// SIMATIC STEP 7 (V5.x) project PROJECT-PROFIBUS_en
// CPU: CPU 314(1)
// CPU: CPU 314(1)
// CPU: CPU 314(1)
// CPU: CPU 314(1)
// CPU: CPU 314(1)
// CPU: CPU 414-2 DP(1)
// CPU: CPU 414-2 DP(1)
// station: P_ADR_BUS
// station: Hardware
// station: FMS-Server S7 400-Stat.
// station: P_ADR_BUS
// station: Hardware
// station: SIMATIC 300-Station(1)
// station: P_ADR_BUS
// station: Hardware
// station: SIMATIC 300-Station(3)
// station: P_ADR_BUS
// station: Hardware
// station: SIMATIC 300 DP-Slave
// station: P_ADR_BUS
// station: Hardware
// station: FMS-Client S7 400-Stat.
// station: P_ADR_BUS
// station: Hardware
// station: SIMATIC 300-Station(2)
// station: P_ADR_BUS
// station: Hardware
// station: SIMATIC 300 DP-Master
// station: ISA_LOCAL_ADR_BUS
// program: S7 Programm (6)
// program: S7 Program (3)
// program: S7 Program(2)
// program: S7 Program (5)
// program: S7 Program (7)
// program: S7 Program (4)
// program: S7 Program(1)

SYMBOL_TABLE
"Index100 READ parameters"	DB 100	DB 100	// READ parameters
"Index101 READ parameters"	DB 101	DB 101	// READ parameters
"Index102 READ parameters"	DB 102	DB 102	// READ parameters
"Index100 WRITE parameter"	DB 200	DB 200	// WRITE parameters
"Index101 WRITE parameter"	DB 201	DB 201	// WRITE parameters
"Index102 WRITE parameter"	DB 202	DB 202	// WRITE parameters
"Index100 Variable dest"	DB 500	DB 500	// Variable destination
"Index101 Variable dest"	DB 501	DB 501	// Variable destination
"Index102 Variable dest"	DB 502	DB 502	// Variable destination
"Index100 Variable source"	DB 600	DB 600	// Variable source
"Index101 Variable source"	DB 601	DB 601	// Variable source
"Index102 Variable source"	DB 602	DB 602	// Variable source
"IDENT"	FB 2	FB 2	// FMS IDENT
"READ"	FB 3	FB 3	// Read function block for FMS services with SIMATIC NET CPs
"WRITE"	FB 6	FB 6	// Write function block for FMS services with SIMATIC NET CPs
"Index100 READ call"	FC 100	FC 100	// READ call
"Index101 READ call"	FC 101	FC 101	// READ call
"Index102 READ call"	FC 102	FC 102	// READ call
"Index100 WRITE call"	FC 200	FC 200	// WRITE call
"Index101 WRITE call"	FC 201	FC 201	// WRITE call
"Index102 WRITE call"	FC 202	FC 202	// WRITE call
"Compare Index 100"	FC 300	FC 300	// Compare index 100
"Error check"	M 0.0	BOOL	// Error check
"BSEND"	SFB 12	SFB 12	// Block-oriented send
"BRCV"	SFB 13	SFB 13	// Block-oriented receive
"BLKMOV"	SFC 20	SFC 20	// Direct word move
"TEST_DB"	SFC 24	SFC 24	// Debug data block
"CONTROL"	SFC 62	SFC 62	// Control status of a CFB instance
"observe Read/Write"	VAT 1		// Monitor read/write
"observe variables"	VAT 2		// Monitor variables
END_SYMBOL_TABLE

// FB 3: know-how protected block, not included

// FB 6: know-how protected block, not included

FUNCTION "Index100 READ call" : VOID	// FC 100
TITLE = CALL_READ
//This function illustrates an FMS communication job with the READ (FB3) function 
//block. A variable of the type integer is accessed.
VERSION : 0.1
BEGIN
NETWORK
TITLE = Read variable with index 100. 
//Read data access:   
//A variable with index 100 is read and entered in the destination data area 
//(here 
//DB500).
//Call parameters in DB 100.
//
//Job handling /job coordination:
//This job is only started when all other jobs have been completed. This means 
//that access to the variable is synchronized.
//The job is triggered by a signal edge at the REQ input. REQ is reset when the 
//job is completed or an error occurred. Following this, the signal is set again.
//If an error occurred, the error number can be read from the status word.
//*
//Only execute job when no other job is active.
      O     "Index100 WRITE parameter".Write_REQ;	//  REQ=1, WRITE is still active
      O     "Index101 READ parameters".Read_REQ;	//    REQ=1, READ is still active
      O     "Index101 WRITE parameter".Write_REQ;	//  REQ=1, WRITE is still active
      O     "Index102 READ parameters".Read_REQ;	//    REQ=1, READ is still active
      O     "Index102 WRITE parameter".Write_REQ;	//  REQ=1, WRITE is still active
      JC    ende;
//*
//Calling the READ job:                                       
//*
//*
//Query job status
//*
//*
//*
//Error handling
//*
      CALL  "READ" , DB 300 (
           DIX 0.0                  := "Index100 READ parameters".Read_REQ,
           DID 2                    := "Index100 READ parameters".Read_ID,
           DIW 6                    := W#16#1002,
           DIW 8                    := 7,
           DIW 10                   := 100,
           DID 12                   := P#DBX 6.0,
           DIW 16                   := W#16#1005,
           DIW 18                   := 1,
           DIW 20                   := 500,
           DID 22                   := P#DBX 0.0,
           DIX 26.0                 := "Index100 READ parameters".Read_NDR,
           DIX 26.1                 := "Index100 READ parameters".Read_Error,
           DIW 28                   := "Index100 READ parameters".Read_Status);	//  REQ=1 => Job active, query errors  /   REQ=1 => Job completed  /   Set REQ again /  Error=0 => No error occurred
      A     "Index100 READ parameters".Read_REQ;
//*
      JC    fehl;	// Error=1 => Error occurred 
      AN    "Index100 READ parameters".Read_REQ;	//Load error status
      S     "Index100 READ parameters".Read_REQ;	// Save in buffer
      JU    ende;	//   Reset REQ
fehl: AN    "Index100 READ parameters".Read_Error;
//*
//Query job status
//*
      JC    ok;	//  Done=0 => Job still active
      A     "Index100 READ parameters".Read_Error;
//*
      L     "Index100 READ parameters".Read_Status;	//  Done=1 => Job complete without error
      T     "Index100 READ parameters".Read_Statusmemory;	//  Reset REQ
//*
      R     "Index100 READ parameters".Read_REQ;
      JU    ende;
ok:   AN    "Index100 READ parameters".Read_NDR;
      JC    ende;
      A     "Index100 READ parameters".Read_NDR;
      R     "Index100 READ parameters".Read_REQ;
ende: BE;
END_FUNCTION

FUNCTION "Index101 READ call" : VOID	// FC 101
TITLE = CALL_READ
//The function illustrates an FMS communication job with the READ (FB3) function 
//block. A variable of the type array is accessed.
VERSION : 0.1
BEGIN
NETWORK
TITLE = Read variable with index 101. 
//Read data access:
//The variable with index 101 is read and entered in the destination data area 
//(here DB501). Call parameters in DB101.
//
//Job handling /job coordination:
//This job is only started when all other jobs have been completed. This means 
//that access to the variable is synchronized.
//The job is triggered by a signal edge at the REQ input. REQ is reset when the 
//job is completed or an error occurred. Following this, the signal is set again.
//If an error occurred, the error number can be read from the status word.
//
//*
// Only execute job when no other job is active.
//*
      O     "Index100 WRITE parameter".Write_REQ;	//  REQ=1, WRITE is still active
      O     "Index100 READ parameters".Read_REQ;	//    REQ=1, READ is still active
      O     "Index101 WRITE parameter".Write_REQ;	//  REQ=1, WRITE is still active
      O     "Index102 READ parameters".Read_REQ;	//    REQ=1, READ is still active
      O     "Index102 WRITE parameter".Write_REQ;	//  REQ=1, WRITE is still active
      JC    ende;
//*
//Calling the READ job:                                       
//*
//*
//Query job status
//*
//*
//*
//Error handling
//*
      CALL  "READ" , DB 301 (
           DIX 0.0                  := "Index101 READ parameters".Read_REQ,
           DID 2                    := "Index101 READ parameters".Read_ID,
           DIW 6                    := W#16#1002,
           DIW 8                    := 7,
           DIW 10                   := 101,
           DID 12                   := P#DBX 6.0,
           DIW 16                   := W#16#1002,
           DIW 18                   := 10,
           DIW 20                   := 501,
           DID 22                   := P#DBX 0.0,
           DIX 26.0                 := "Index101 READ parameters".Read_NDR,
           DIX 26.1                 := "Index101 READ parameters".Read_Error,
           DIW 28                   := "Index101 READ parameters".Read_Status);	//   REQ=1 => Job active, query errors /    REQ=1 => Job completed /    REQ neu setzten / Set REQ again /  Error=0 => No error occurred
      A     "Index101 READ parameters".Read_REQ;
//*
      JC    fehl;	// Error=1 => Error occurred
      AN    "Index101 READ parameters".Read_REQ;	// load error status
      S     "Index101 READ parameters".Read_REQ;	// Save in buffer
      JU    ende;	//   Reset REQ
fehl: AN    "Index101 READ parameters".Read_Error;
//*
//Query job status
//*
      JC    ok;	//  Done=0 => Job still active
      A     "Index101 READ parameters".Read_Error;
//*
      L     "Index101 READ parameters".Read_Status;	//  Done=1 => Job complete without error
      T     "Index101 READ parameters".Read_Statusspeicher;	//  Reset REQ
//*
      R     "Index101 READ parameters".Read_REQ;
      JU    ende;
ok:   AN    "Index101 READ parameters".Read_NDR;
      JC    ende;
      A     "Index101 READ parameters".Read_NDR;
      R     "Index101 READ parameters".Read_REQ;
ende: BE;
END_FUNCTION

FUNCTION "Index102 READ call" : VOID	// FC 102
TITLE = CALL_READ
//This function illustrates an FMS communication job with the READ (FB3) function 
//block. A variable of the type STRUCT is accessed.
VERSION : 0.1
BEGIN
NETWORK
TITLE = Read variable with index 102.
//Read data access:   
//A variable with index 102 is read and entered in the destination data area 
//(here 
//DB502). Call parameters in DB 100.
//
//Job handling /job coordination:
//This job is only started when all other jobs have been completed. This means 
//that access to the variable is synchronized.
//The job is triggered by a signal edge at the REQ input. REQ is reset when the 
//job is completed or an error occurred. Following this, the signal is set again.
//If an error occurred, the error number can be read from the status word.
//*
// Query whether other jobs still active
//*
      O     "Index100 READ parameters".Read_REQ;	//    REQ=1, READ is still active
      O     "Index100 WRITE parameter".Write_REQ;	//  REQ=1, WRITE is still active
      O     "Index101 READ parameters".Read_REQ;	//    REQ=1, READ is still active
      O     "Index101 WRITE parameter".Write_REQ;	//  REQ=1, WRITE is still active
      O     "Index102 WRITE parameter".Write_REQ;	//  REQ=1, WRITEis still active
      JC    ende;
//*
// Calling the READ job                                      
//*
//*
// Query the job status
//*
//*
//*
// Error handling
//*
      CALL  "READ" , DB 302 (
           DIX 0.0                  := "Index102 READ parameters".Read_REQ,
           DID 2                    := "Index102 READ parameters".Read_ID,
           DIW 6                    := W#16#1002,
           DIW 8                    := 7,
           DIW 10                   := 102,
           DID 12                   := P#DBX 6.0,
           DIW 16                   := W#16#1002,
           DIW 18                   := 18,
           DIW 20                   := 502,
           DID 22                   := P#DBX 0.0,
           DIX 26.0                 := "Index102 READ parameters".Read_NDR,
           DIX 26.1                 := "Index102 READ parameters".Read_Error,
           DIW 28                   := "Index102 READ parameters".Read_Status);	//   REQ=1 => Job active, query errors /    REQ=1 => Job completed /    Set REQ again /  Error=0 => No error occurred
      A     "Index102 READ parameters".Read_REQ;
//*
      JC    fehl;	//  Error=1 => Error occurred
      AN    "Index102 READ parameters".Read_REQ;	// Load error status
      S     "Index102 READ parameters".Read_REQ;	// Save in buffer
      JU    ende;	//  Reset REQ
fehl: AN    "Index102 READ parameters".Read_Error;
//*
// Query job status
//*
      JC    ok;	//  Done=0 => Job still active
      A     "Index102 READ parameters".Read_Error;
//*
      L     "Index102 READ parameters".Read_Status;	// Done=1 => Job complete without error
      T     "Index102 READ parameters".Read_Statusspeicher;	//   Reset REQ
//*
      R     "Index102 READ parameters".Read_REQ;
      JU    ende;
ok:   AN    "Index102 READ parameters".Read_NDR;
      JC    ende;
      A     "Index102 READ parameters".Read_NDR;
      R     "Index102 READ parameters".Read_REQ;
ende: BE;
END_FUNCTION

FUNCTION "Index100 WRITE call" : VOID	// FC 200
TITLE = CALL_WRITE
//This function illustrates an FMS communication job with the WRITE (FB6) 
//function 
//block. A variable of the type integer is accessed.
VERSION : 0.1
BEGIN
NETWORK
TITLE = Write var. with index 100 
//Write data access:   
//A variable with index 100 is written. It is taken from the source data area 
//(here DB600). Call parameters in DB200.
//
//Job handling /job coordination:
//This job is only started when all other jobs have been completed. This means 
//that access to the variable is synchronized.
//The job is triggered by a signal edge at the REQ input. REQ is reset when the 
//job is completed or an error occurred. Following this, the signal is set again.
//If an error occurred, the error number can be read from the status word.
//
//*  
// Query whether other jobs active
//*
      O     "Index100 READ parameters".Read_REQ;	//    REQ=1, WRITE is still active
      O     "Index101 READ parameters".Read_REQ;	//    REQ=1, READ is still active
      O     "Index101 WRITE parameter".Write_REQ;	//  REQ=1, WRITE is still active
      O     "Index102 READ parameters".Read_REQ;	//    REQ=1, READ is still active
      O     "Index102 WRITE parameter".Write_REQ;	//  REQ=1, WRITE is still active
      JC    ende;
//*
// Calling the write job               
//*
//*
// Query the job status
//*
//*
// *
// Error handling
//*
      CALL  "WRITE" , DB 400 (
           DIX 0.0                  := "Index100 WRITE parameter".Write_REQ,
           DID 2                    := "Index100 WRITE parameter".Write_ID,
           DIW 6                    := W#16#1002,
           DIW 8                    := 7,
           DIW 10                   := 200,
           DID 12                   := P#DBX 6.0,
           DIW 16                   := W#16#1005,
           DIW 18                   := 1,
           DIW 20                   := 600,
           DID 22                   := P#DBX 0.0,
           DIX 26.0                 := "Index100 WRITE parameter".Write_Done,
           DIX 26.1                 := "Index100 WRITE parameter".Write_Error,
           DIW 28                   := "Index100 WRITE parameter".Write_Status);	//    REQ=1 => Job active, query errors /     REQ=1 => Job completed  /     Set REQ again /   Error=0 => No error occurred
      A     "Index100 WRITE parameter".Write_REQ;
//*
      JC    fehl;	//  Error=1 => Error occurred
      AN    "Index100 WRITE parameter".Write_REQ;	// Load error status
      S     "Index100 WRITE parameter".Write_REQ;	// Save in buffer
      JU    ende;	//    Reset REQ
fehl: AN    "Index100 WRITE parameter".Write_Error;
//*
// Query job status 
//*
      JC    ok;	//   Done=0 => Job still active
      A     "Index100 WRITE parameter".Write_Error;
//*
      L     "Index100 WRITE parameter".Write_Status;	//   Done=1 => Job complete without error
      T     "Index100 WRITE parameter".Write_Statusspeicher;	//     / Reset REQ
//*
      R     "Index100 WRITE parameter".Write_REQ;
      JU    ende;
ok:   AN    "Index100 WRITE parameter".Write_Done;
      JC    ende;
      A     "Index100 WRITE parameter".Write_Done;
      R     "Index100 WRITE parameter".Write_REQ;
ende: BE;
END_FUNCTION

FUNCTION "Index101 WRITE call" : VOID	// FC 201
TITLE = CALL_WRITE
//This function illustrates an FMS communication job with the WRITE (FB6) 
//function 
//block. A variable of the type ARRAY is accessed.
//
VERSION : 0.1
BEGIN
NETWORK
TITLE = Write var with index 101. 
//Write data access:   
//A variable with index 100 is written. It is taken from the source data area 
//(here DB601). Call parameters in DB201.
//
//Job handling /job coordination:
//This job is only started when all other jobs have been completed. This means 
//that access to the variable is synchronized.
//The job is triggered by a signal edge at the REQ input. REQ is reset when the 
//job is completed or an error occurred. Following this, the signal is set 
//again.
//If an error occurred, the error number can be read from the status word.
//*  
// Query whether other jobs still active
//*
      O     "Index100 READ parameters".Read_REQ;	//    REQ=1, WRITE is still active
      O     "Index100 WRITE parameter".Write_REQ;	//  REQ=1, WRITE is still active
      O     "Index101 READ parameters".Read_REQ;	//    REQ=1, READ is still active
      O     "Index102 READ parameters".Read_REQ;	//    REQ=1, READ is still active
      O     "Index102 WRITE parameter".Write_REQ;	//  REQ=1, WRITE is still active
      JC    ende;
//*
// Calling the write job               
//*
//*
// Query job status
//*
//*
// *
// Error handling
//*
      CALL  "WRITE" , DB 401 (
           DIX 0.0                  := "Index101 WRITE parameter".Write_REQ,
           DID 2                    := "Index101 WRITE parameter".Write_ID,
           DIW 6                    := W#16#1002,
           DIW 8                    := 7,
           DIW 10                   := 201,
           DID 12                   := P#DBX 6.0,
           DIW 16                   := W#16#1002,
           DIW 18                   := 10,
           DIW 20                   := 601,
           DID 22                   := P#DBX 0.0,
           DIX 26.0                 := "Index101 WRITE parameter".Write_Done,
           DIX 26.1                 := "Index101 WRITE parameter".Write_Error,
           DIW 28                   := "Index101 WRITE parameter".Write_Status);	//    REQ=1 => Job active, query errors  /     REQ=1 => Job completed   /     Set REQ again /    Error=0 => No error occurred
      A     "Index101 WRITE parameter".Write_REQ;
//*
      JC    fehl;	//  Error=1 => Error occurred
      AN    "Index101 WRITE parameter".Write_REQ;	// Load error status
      S     "Index101 WRITE parameter".Write_REQ;	// Save in buffer
      JU    ende;	//    Reset REQ
fehl: AN    "Index101 WRITE parameter".Write_Error;
//*
// Query job status
//*
      JC    ok;	//   Done=0 => Job still active
      A     "Index101 WRITE parameter".Write_Error;
//*
      L     "Index101 WRITE parameter".Write_Status;	//   Done=1 => Job complete without error
      T     "Index101 WRITE parameter".Write_Statusspeicher;	//    Reset REQ
//*
      R     "Index101 WRITE parameter".Write_REQ;
      JU    ende;
ok:   AN    "Index101 WRITE parameter".Write_Done;
      JC    ende;
      A     "Index101 WRITE parameter".Write_Done;
      R     "Index101 WRITE parameter".Write_REQ;
ende: BE;
END_FUNCTION

FUNCTION "Index102 WRITE call" : VOID	// FC 202
TITLE = CALL_WRITE
//This function illustrates an FMS communication job with the WRITE (FB6) 
//function 
//block. A variable of the type STRUCT is accessed.
//
VERSION : 0.1
BEGIN
NETWORK
TITLE = Write var with index 102.
//Write data access:   
//A variable with index 102 is written. It is taken from the source data area 
//(here DB602). Call parameters in DB202.
//
//Job handling /job coordination:
//This job is only started when all other jobs have been completed. This means 
//that access to the variable is synchronized.
//The job is triggered by a signal edge at the REQ input. REQ is reset when the 
//job is completed or an error occurred. Following this, the signal is set again.
//If an error occurred, the error number can be read from the status word.
//
//
//*  
// Query whether other jobs active
//*       
      O     "Index100 READ parameters".Read_REQ;	//    REQ=1, READ is still active
      O     "Index100 WRITE parameter".Write_REQ;	//  REQ=1, WRITE is still active
      O     "Index101 READ parameters".Read_REQ;	//    REQ=1, REA is still active
      O     "Index101 WRITE parameter".Write_REQ;	//  REQ=1, WRITE is still active
      O     "Index102 READ parameters".Read_REQ;	//    REQ=1, REA is still active
      JC    ende;
//*
// Calling the write job               
//*
//*
// Query job status
//*
//*
// *
// Error handling
//*
      CALL  "WRITE" , DB 402 (
           DIX 0.0                  := "Index102 WRITE parameter".Write_REQ,
           DID 2                    := "Index102 WRITE parameter".Write_ID,
           DIW 6                    := W#16#1002,
           DIW 8                    := 7,
           DIW 10                   := 202,
           DID 12                   := P#DBX 6.0,
           DIW 16                   := W#16#1002,
           DIW 18                   := 18,
           DIW 20                   := 602,
           DID 22                   := P#DBX 0.0,
           DIX 26.0                 := "Index102 WRITE parameter".Write_Done,
           DIX 26.1                 := "Index102 WRITE parameter".Write_Error,
           DIW 28                   := "Index102 WRITE parameter".Write_Status);	//    REQ=1 => Job active, query errors /     REQ=1 => Job completed /     Set REQ again /   Error=0 => No error occurred
      A     "Index102 WRITE parameter".Write_REQ;
//*
      JC    fehl;	//  Error=1 => Error occurred
      AN    "Index102 WRITE parameter".Write_REQ;	// Load error status
      S     "Index102 WRITE parameter".Write_REQ;	// Save in buffer
      JU    ende;	//    Reset REQ
fehl: AN    "Index102 WRITE parameter".Write_Error;
//*
// Query job status 
//*
      JC    ok;	//   Done=0 => Job still active
      A     "Index102 WRITE parameter".Write_Error;
//*
      L     "Index102 WRITE parameter".Write_Status;	//   Done=1 => Job complete without error
      T     "Index102 WRITE parameter".Write_Statusspeicher;	//    Reset REQ
//*
      R     "Index102 WRITE parameter".Write_REQ;
      JU    ende;
ok:   AN    "Index102 WRITE parameter".Write_Done;
      JC    ende;
      A     "Index102 WRITE parameter".Write_Done;
      R     "Index102 WRITE parameter".Write_REQ;
ende: BE;
END_FUNCTION

FUNCTION "Compare Index 100" : VOID	// FC 300
//This function simulates a signal or value change and checks the write or read 
//function via the FMS connection. 
VERSION : 0.1
BEGIN
NETWORK
TITLE = Error check
//After writing and reading index 100, the values are compared to check that they 
//match. Afterwards the variable is incremented by one.
//
//*
      L     "Index100 Variable dest".Index_100;
      L     "Index100 Variable source".Index_100;
      ==I;
      JC    inkr;
//*
// Set memory bit 0.0 if the source and destination do not match.
//*
      S     "Error check";
//*
// Increment variable with index 100 by one
//*
inkr: L     "Index100 Variable source".Index_100;
      +     1;
      T     "Index100 Variable source".Index_100;
      R     "Error check";
//*
      BE;
END_FUNCTION

DATA_BLOCK "Index100 READ parameters"	// DB 100
VERSION : 0.1
  STRUCT
   Read_REQ : BOOL ;
   Read_ID : DWORD  := DW#16#10001;
   Read_VAR_Index : STRING  [5 ] := '<100>';
   Read_NDR : BOOL ;
   Read_Error : BOOL ;
   Read_Status : WORD ;
   Read_Statusmemory : WORD ;
  END_STRUCT ;	
BEGIN
   Read_ID := DW#16#10001;
   Read_VAR_Index := '<100>';
END_DATA_BLOCK

DATA_BLOCK "Index101 READ parameters"	// DB 101
VERSION : 0.1
  STRUCT
   Read_REQ : BOOL ;
   Read_ID : DWORD  := DW#16#10001;
   Read_VAR_Index : STRING  [5 ] := '<101>';
   Read_NDR : BOOL ;
   Read_Error : BOOL ;
   Read_Status : WORD ;
   Read_Statusspeicher : WORD ;
  END_STRUCT ;	
BEGIN
   Read_ID := DW#16#10001;
   Read_VAR_Index := '<101>';
END_DATA_BLOCK

DATA_BLOCK "Index102 READ parameters"	// DB 102
VERSION : 0.1
  STRUCT
   Read_REQ : BOOL ;
   Read_ID : DWORD  := DW#16#10001;
   Read_VAR_Index : STRING  [5 ] := '<102>';
   Read_NDR : BOOL ;
   Read_Error : BOOL ;
   Read_Status : WORD ;
   Read_Statusspeicher : WORD ;
  END_STRUCT ;	
BEGIN
   Read_ID := DW#16#10001;
   Read_VAR_Index := '<102>';
END_DATA_BLOCK

DATA_BLOCK "Index100 WRITE parameter"	// DB 200
VERSION : 0.1
  STRUCT
   Write_REQ : BOOL ;
   Write_ID : DWORD  := DW#16#10001;
   Write_VAR_Index : STRING  [5 ] := '<100>';
   Write_Done : BOOL ;
   Write_Error : BOOL ;
   Write_Status : WORD ;
   Write_Statusspeicher : WORD ;
   Write_VAR_Index1 : STRING  [5 ] := '<100>';
   tdmset : BYTE ;
  END_STRUCT ;	
BEGIN
   Write_ID := DW#16#10001;
   Write_VAR_Index := '<100>';
   Write_VAR_Index1 := '<100>';
END_DATA_BLOCK

DATA_BLOCK "Index101 WRITE parameter"	// DB 201
VERSION : 0.1
  STRUCT
   Write_REQ : BOOL ;
   Write_ID : DWORD  := DW#16#10001;
   Write_VAR_Index : STRING  [5 ] := '<101>';
   Write_Done : BOOL ;
   Write_Error : BOOL ;
   Write_Status : WORD ;
   Write_Statusspeicher : WORD ;
  END_STRUCT ;	
BEGIN
   Write_ID := DW#16#10001;
   Write_VAR_Index := '<101>';
END_DATA_BLOCK

DATA_BLOCK "Index102 WRITE parameter"	// DB 202
VERSION : 0.1
  STRUCT
   Write_REQ : BOOL ;
   Write_ID : DWORD  := DW#16#10001;
   Write_VAR_Index : STRING  [5 ] := '<102>';
   Write_Done : BOOL ;
   Write_Error : BOOL ;
   Write_Status : WORD ;
   Write_Statusspeicher : WORD ;
  END_STRUCT ;	
BEGIN
   Write_ID := DW#16#10001;
   Write_VAR_Index := '<102>';
END_DATA_BLOCK

DATA_BLOCK DB 300
AUTHOR : SIMATIC
FAMILY : CP_400
VERSION : 0.0
"READ"
BEGIN
END_DATA_BLOCK

DATA_BLOCK DB 301
AUTHOR : SIMATIC
FAMILY : CP_400
VERSION : 0.0
"READ"
BEGIN
END_DATA_BLOCK

DATA_BLOCK DB 302
AUTHOR : SIMATIC
FAMILY : CP_400
VERSION : 0.0
"READ"
BEGIN
END_DATA_BLOCK

DATA_BLOCK DB 400
AUTHOR : SIMATIC
FAMILY : CP_400
VERSION : 0.0
"WRITE"
BEGIN
END_DATA_BLOCK

DATA_BLOCK DB 401
AUTHOR : SIMATIC
FAMILY : CP_400
VERSION : 0.0
"WRITE"
BEGIN
END_DATA_BLOCK

DATA_BLOCK DB 402
AUTHOR : SIMATIC
FAMILY : CP_400
VERSION : 0.0
"WRITE"
BEGIN
END_DATA_BLOCK

DATA_BLOCK "Index100 Variable dest"	// DB 500
VERSION : 0.1
  STRUCT
   Index_100 : INT ;
  END_STRUCT ;	
BEGIN
END_DATA_BLOCK

DATA_BLOCK "Index101 Variable dest"	// DB 501
VERSION : 0.1
  STRUCT
   Index_101 : ARRAY  [1 .. 10 ] OF BYTE ;
  END_STRUCT ;	
BEGIN
END_DATA_BLOCK

DATA_BLOCK "Index102 Variable dest"	// DB 502
VERSION : 0.1
  STRUCT
   Index_102 : STRUCT
    Subindex_1 : BOOL ;
    Subindex_2 : STRING  [8 ];
    Subindex_3 : CHAR ;
    Subindex_4 : DINT ;
   END_STRUCT ;
  END_STRUCT ;	
BEGIN
   Index_102.Subindex_3 := ' ';
END_DATA_BLOCK

DATA_BLOCK "Index100 Variable source"	// DB 600
VERSION : 0.1
  STRUCT
   Index_100 : INT ;
  END_STRUCT ;	
BEGIN
END_DATA_BLOCK

DATA_BLOCK "Index101 Variable source"	// DB 601
VERSION : 0.1
  STRUCT
   Index_101 : ARRAY  [1 .. 10 ] OF BYTE ;
  END_STRUCT ;	
BEGIN
END_DATA_BLOCK

DATA_BLOCK "Index102 Variable source"	// DB 602
VERSION : 0.1
  STRUCT
   Index_102 : STRUCT
    Subindex_1 : BOOL ;
    Subindex_2 : STRING  [8 ] := 'Hello!!!';
    Subindex_3 : CHAR ;
    Subindex_4 : DINT ;
   END_STRUCT ;
  END_STRUCT ;	
BEGIN
   Index_102.Subindex_2 := 'Andreas!';
   Index_102.Subindex_3 := ' ';
END_DATA_BLOCK

ORGANIZATION_BLOCK OB 1
//Functions (FC100..FC300) in which FMS communication jobs are sent are called in 
//this block. The FCs are designed so that a coordinated sequence is guaranteed.
//(For the symbolic declaration, refer to the entries in the symbol table for 
//this 
//CPU.)
VERSION : 0.1
VAR_TEMP
  OB1_EV_CLASS : BYTE ;	//Bits 0-3 = 1 (Coming event), Bits 4-7 = 1 (Event class 1)
  OB1_SCAN_1 : BYTE ;	//1 (Cold restart scan 1 of OB 1), 3 (Scan 2-n of OB 1)
  OB1_PRIORITY : BYTE ;	//1 (Priority of 1 is lowest)
  OB1_OB_NUMBR : BYTE ;	//1 (Organization block 1, OB1)
  OB1_RESERVED_1 : BYTE ;	//Reserved for system
  OB1_RESERVED_2 : BYTE ;	//Reserved for system
  OB1_PREV_CYCLE : INT ;	//Cycle time of previous OB1 scan (milliseconds)
  OB1_MIN_CYCLE : INT ;	//Minimum cycle time of OB1 (milliseconds)
  OB1_MAX_CYCLE : INT ;	//Maximum cycle time of OB1 (milliseconds)
  OB1_DATE_TIME : DATE_AND_TIME ;	//Date and time OB1 started
END_VAR
BEGIN
NETWORK
TITLE =
//Write and read jobs are called sequentially.
      CALL  "Index100 READ call";
//*
      CALL  "Compare Index 100";
//*
      CALL  "Index100 WRITE call";
//*
      CALL  "Index101 READ call";
//*
      CALL  "Index101 WRITE call";
//*
      CALL  "Index102 READ call";
//*
      CALL  "Index102 WRITE call";
END_ORGANIZATION_BLOCK

ORGANIZATION_BLOCK OB 100
VERSION : 0.1
VAR_TEMP
  OB100_EV_CLASS : BYTE ;	//16#13, Event class 1, Entering event state, Event logged in diagnostic buffer
  OB100_STRTUP : BYTE ;	//16#81/82/83/84 Method of startup
  OB100_PRIORITY : BYTE ;	//27 (Priority of 1 is lowest)
  OB100_OB_NUMBR : BYTE ;	//100 (Organization block 100, OB100)
  OB100_RESERVED_1 : BYTE ;	//Reserved for system
  OB100_RESERVED_2 : BYTE ;	//Reserved for system
  OB100_STOP : WORD ;	//Event that caused CPU to stop (16#4xxx)
  OB100_STRT_INFO : DWORD ;	//Information on how system started
  OB100_DATE_TIME : DATE_AND_TIME ;	//Date and time OB100 started
END_VAR
BEGIN
NETWORK
TITLE =
      L     0;
      T     "Index100 Variable dest".Index_100;
      BE;
END_ORGANIZATION_BLOCK

SYMBOL_TABLE
"DP_SEND"	FC 1	FC 1	// DP SEND
"DP_RECV"	FC 2	FC 2	// DP RECEIVE
"DP_DIAG"	FC 3	FC 3	// DP DIAGNOSE
"DP_CTRL"	FC 4	FC 4	// DP CONTROL
"STP"	SFC 46	SFC 46	// Change the CPU to STOP
"WR_REC"	SFC 58	SFC 58	// Write Data Record
"RD_REC"	SFC 59	SFC 59	// Read a Data Record
END_SYMBOL_TABLE

// FC 1: know-how protected block, not included

// FC 2: know-how protected block, not included

// FC 3: know-how protected block, not included

// FC 4: know-how protected block, not included

FUNCTION FC 29 : VOID
TITLE = running light
VERSION : 0.1
BEGIN
NETWORK
TITLE =
      A     T 4;	//time downwards
      JC    runt;
st_1: A     M 40.1;	//start timer 3
      L     S5T#3S;	//LED upwards 3 sec.
      SE    T 3;
      A     T 3;
      R     M 40.1;
      JC    hoch;	//jump to upwards
      AN    T 3;
      S     M 40.1;
      S     M 40.2;
runt: A     M 40.2;	//start timer 4
      L     S5T#3S;	//LED downwards 3 sec.
      SE    T 4;
      A     T 4;
      R     M 40.2;
      AN    T 4;
      S     M 40.2;
      JC    st_1;
      A     M 40.0;
      L     S5T#100MS;
      SE    T 1;
      A     T 1;
      R     M 40.0;
      A     T 1;
      JC    weit;
      AN    T 1;
      S     M 40.0;
      L     MW 70;
      L     0;
      <>D;
      JC    los1;
      TAK;
      +     1;
      T     MW 70;
      T     DB30.DBW 1;
      BEU;
los1: L     MW 70;
      L     2;
      *D;
      T     MW 70;
      T     DB30.DBW 1;
      L     L#32768;
      <>D;
      BEC;
      L     0;
      T     MW 70;
weit: BEU;
hoch: A     M 40.3;
      L     S5T#100MS;
      SE    T 1;
      A     T 1;
      R     M 40.3;
      A     T 1;
      JC    weit;
      AN    T 1;
      S     M 40.3;
      L     MW 70;
      L     0;
      <>D;
      JC    los2;
      TAK;
      +     L#32768;
      T     MW 70;
      T     DB30.DBW 1;
      BEU;
los2: L     MW 70;
      L     2;
      /D;
      T     MW 70;
      T     DB30.DBW 1;
      L     1;
      <>D;
      BEC;
      L     0;
      T     MW 70;
      BE;
END_FUNCTION

ORGANIZATION_BLOCK OB 1
TITLE = co-ordination DP-Slave
//Co-ordination of the program sequence.
VERSION : 0.1
VAR_TEMP
  OB1_EV_CLASS : BYTE ;	//Bits 0-3 = 1 (Coming event), Bits 4-7 = 1 (Event class 1)
  OB1_SCAN_1 : BYTE ;	//1 (Cold restart scan 1 of OB 1), 3 (Scan 2-n of OB 1)
  OB1_PRIORITY : BYTE ;	//1 (Priority of 1 is lowest)
  OB1_OB_NUMBR : BYTE ;	//1 (Organization block 1, OB1)
  OB1_RESERVED_1 : BYTE ;	//Reserved for system
  OB1_RESERVED_2 : BYTE ;	//Reserved for system
  OB1_PREV_CYCLE : INT ;	//Cycle time of previous OB1 scan (milliseconds)
  OB1_MIN_CYCLE : INT ;	//Minimum cycle time of OB1 (milliseconds)
  OB1_MAX_CYCLE : INT ;	//Maximum cycle time of OB1 (milliseconds)
  OB1_DATE_TIME : DATE_AND_TIME ;	//Date and time OB1 started
END_VAR
BEGIN
NETWORK
TITLE =
      CALL  "DP_RECV" (
           $1                       := 272,
           $2                       := P#DB10.DBX 0.0 BYTE 10,
           $3                       := P#M 1.0,
           $4                       := M 1.1,
           $5                       := P#M 200.0,
           $6                       := P#M 202.0);	//Call DP_RECV
      L     DB10.DBW 0;	//output for simulation module
      T     QW 0;
      T     DB11.DBW 0;	//data for confirmation
      CALL  "DP_SEND" (
           $1                       := 272,
           $2                       := P#DB11.DBX 0.0 BYTE 10,
           $3                       := M 1.2,
           $4                       := M 1.3,
           $5                       := P#M 104.0);	//Call DP_SEND
      BE;
END_ORGANIZATION_BLOCK

ORGANIZATION_BLOCK OB 100
TITLE = create DB
//Creation of data blocks DB10 and DB11. The process values are saved in these 
//data blocks.
VERSION : 0.0
VAR_TEMP
  OB100_EV_CLASS : BYTE ;	//16#13, Event class 1, Entering event state, Event logged in diagnostic buffer
  OB100_STRTUP : BYTE ;	//16#81/82/83/84 Method of startup
  OB100_PRIORITY : BYTE ;	//27 (Priority of 1 is lowest)
  OB100_OB_NUMBR : BYTE ;	//100 (Organization block 100, OB100)
  OB100_RESERVED_1 : BYTE ;	//Reserved for system
  OB100_RESERVED_2 : BYTE ;	//Reserved for system
  OB100_STOP : WORD ;	//Event that caused CPU to stop (16#4xxx)
  OB100_STRT_INFO : DWORD ;	//Information on how system started
  OB100_DATE_TIME : DATE_AND_TIME ;	//Date and time OB100 started
END_VAR
BEGIN
NETWORK
TITLE =
      L     10;
      T     MW 20;
      L     11;
      T     MW 22;
      L     300;
      T     MW 24;
      CALL  SFC 22 (
           LOW_LIMIT                := MW 20,
           UP_LIMIT                 := MW 22,
           COUNT                    := MW 24,
           RET_VAL                  := MW 26,
           DB_NUMBER                := MW 26);
      CALL  SFC 22 (
           LOW_LIMIT                := MW 20,
           UP_LIMIT                 := MW 22,
           COUNT                    := MW 24,
           RET_VAL                  := MW 26,
           DB_NUMBER                := MW 28);
      BE;
END_ORGANIZATION_BLOCK

SYMBOL_TABLE
"AG_SEND"	FC 5	FC 5	// AG SEND
"AG_RECV"	FC 6	FC 6	// AG RECEIVE
END_SYMBOL_TABLE

// FC 5: know-how protected block, not included

// FC 6: know-how protected block, not included

FUNCTION FC 29 : VOID
TITLE = handling of the process data
//A data word is incremented and decremented cyclically. The time interval for 
//incrementing and decrementing is 3 seconds.
VERSION : 0.1
BEGIN
NETWORK
TITLE =
      A     T 4;	//time downwards
      JC    runt;
st_1: A     M 40.1;	//start timer 3
      L     S5T#3S;	//LED upwards 3 sec
      SE    T 3;
      A     T 3;
      R     M 40.1;
      JC    hoch;	//jump for upwards
      AN    T 3;
      S     M 40.1;
      S     M 40.2;
runt: A     M 40.2;	//start timer 4
      L     S5T#3S;	//LED downwards 3 sec
      SE    T 4;
      A     T 4;
      R     M 40.2;
      AN    T 4;
      S     M 40.2;
      JC    st_1;
      A     M 40.0;
      L     S5T#100MS;
      SE    T 1;
      A     T 1;
      R     M 40.0;
      A     T 1;
      JC    weit;
      AN    T 1;
      S     M 40.0;
      L     MW 70;
      L     0;
      <>D;
      JC    los1;
      TAK;
      +     1;
      T     MW 70;
      T     DB30.DBW 1;
      BEU;
los1: L     MW 70;
      L     2;
      *D;
      T     MW 70;
      T     DB30.DBW 1;
      L     L#32768;
      <>D;
      BEC;
      L     0;
      T     MW 70;
weit: BEU;
hoch: A     M 40.3;
      L     S5T#100MS;
      SE    T 1;
      A     T 1;
      R     M 40.3;
      A     T 1;
      JC    weit;
      AN    T 1;
      S     M 40.3;
      L     MW 70;
      L     0;
      <>D;
      JC    los2;
      TAK;
      +     L#32768;
      T     MW 70;
      T     DB30.DBW 1;
      BEU;
los2: L     MW 70;
      L     2;
      /D;
      T     MW 70;
      T     DB30.DBW 1;
      L     1;
      <>D;
      BEC;
      L     0;
      T     MW 70;
      BE;
END_FUNCTION

FUNCTION FC 30 : VOID
TITLE = Senden
//Sends data via FDL-connection with ID=1.
//Starting at byte 1 from DB30, 4 bytes are going to send.
VERSION : 0.0
BEGIN
NETWORK
TITLE =
      O     M 50.0;
      ON    M 50.0;
      S     M 50.0;
      CALL  "AG_SEND" (
           $1                       := P#M 50.0,
           $2                       := 1,
           $3                       := 272,
           $4                       := P#DB30.DBX 1.0 BYTE 240,
           $5                       := 4,
           $6                       := M 1.2,
           $7                       := M 1.3,
           $8                       := P#M 200.0);	//AG_SEND
      BE;
END_FUNCTION

FUNCTION FC 31 : VOID
TITLE = Receive
//Station 1
//
//Receives data via FDL-connection with ID=1.
//Data are accepted in DB31.
VERSION : 0.0
BEGIN
NETWORK
TITLE =
      CALL  "AG_RECV" (
           $1                       := 1,
           $2                       := 272,
           $3                       := P#DB31.DBX 1.0 BYTE 240,
           $4                       := P#M 1.0,
           $5                       := M 1.1,
           $6                       := P#M 202.0,
           $7                       := P#M 10.0);	//AG_RECV
      L     DB31.DBW 1;
      T     QW 0;
      BE;
END_FUNCTION

ORGANIZATION_BLOCK OB 1
TITLE = co-ordination
//Co-ordination of the program sequence.
VERSION : 0.1
VAR_TEMP
  OB1_EV_CLASS : BYTE ;	//Bits 0-3 = 1 (Coming event), Bits 4-7 = 1 (Event class 1)
  OB1_SCAN_1 : BYTE ;	//1 (Cold restart scan 1 of OB 1), 3 (Scan 2-n of OB 1)
  OB1_PRIORITY : BYTE ;	//1 (Priority of 1 is lowest)
  OB1_OB_NUMBR : BYTE ;	//1 (Organization block 1, OB1)
  OB1_RESERVED_1 : BYTE ;	//Reserved for system
  OB1_RESERVED_2 : BYTE ;	//Reserved for system
  OB1_PREV_CYCLE : INT ;	//Cycle time of previous OB1 scan (milliseconds)
  OB1_MIN_CYCLE : INT ;	//Minimum cycle time of OB1 (milliseconds)
  OB1_MAX_CYCLE : INT ;	//Maximum cycle time of OB1 (milliseconds)
  OB1_DATE_TIME : DATE_AND_TIME ;	//Date and time OB1 started
END_VAR
BEGIN
NETWORK
TITLE =
      CALL  FC 29;
      CALL  FC 30;
      CALL  FC 31;
      BE;
END_ORGANIZATION_BLOCK

ORGANIZATION_BLOCK OB 100
TITLE = Create DB
//Creation of data blocks DB30/DB31 with length 350 byte. The process values are 
//saved 
//in these data blocks.
VERSION : 0.0
VAR_TEMP
  OB100_EV_CLASS : BYTE ;	//16#13, Event class 1, Entering event state, Event logged in diagnostic buffer
  OB100_STRTUP : BYTE ;	//16#81/82/83/84 Method of startup
  OB100_PRIORITY : BYTE ;	//27 (Priority of 1 is lowest)
  OB100_OB_NUMBR : BYTE ;	//100 (Organization block 100, OB100)
  OB100_RESERVED_1 : BYTE ;	//Reserved for system
  OB100_RESERVED_2 : BYTE ;	//Reserved for system
  OB100_STOP : WORD ;	//Event that caused CPU to stop (16#4xxx)
  OB100_STRT_INFO : DWORD ;	//Information on how system started
  OB100_DATE_TIME : DATE_AND_TIME ;	//Date and time OB100 started
END_VAR
BEGIN
NETWORK
TITLE =
      L     30;
      T     MW 22;
      L     31;
      T     MW 24;
      L     350;
      T     MW 26;
      CALL  SFC 22 (
           LOW_LIMIT                := MW 22,
           UP_LIMIT                 := MW 24,
           COUNT                    := MW 26,
           RET_VAL                  := MW 28,
           DB_NUMBER                := MW 30);
      BE;
END_ORGANIZATION_BLOCK

SYMBOL_TABLE
"AG_SEND"	FC 5	FC 5	// AG SEND
"AG_RECV"	FC 6	FC 6	// AG RECEIVE
END_SYMBOL_TABLE

// FC 5: know-how protected block, not included

// FC 6: know-how protected block, not included

FUNCTION FC 29 : VOID
TITLE = handling of the process data
//A data word is incremented and decremented cyclically. The time interval for 
//incrementing and decrementing is 3 seconds.
VERSION : 0.1
BEGIN
NETWORK
TITLE =
      A     T 4;	//Time downwards
      JC    runt;
st_1: A     M 40.1;	//start timer 3
      L     S5T#3S;	//LED upwards 3 sec
      SE    T 3;
      A     T 3;
      R     M 40.1;
      JC    hoch;	//jump for upwards
      AN    T 3;
      S     M 40.1;
      S     M 40.2;
runt: A     M 40.2;	//start für timer 4
      L     S5T#3S;	//LED downwards 3 sec
      SE    T 4;
      A     T 4;
      R     M 40.2;
      AN    T 4;
      S     M 40.2;
      JC    st_1;
      A     M 40.0;
      L     S5T#100MS;
      SE    T 1;
      A     T 1;
      R     M 40.0;
      A     T 1;
      JC    weit;
      AN    T 1;
      S     M 40.0;
      L     MW 70;
      L     0;
      <>D;
      JC    los1;
      TAK;
      +     1;
      T     MW 70;
      T     DB30.DBW 1;
      BEU;
los1: L     MW 70;
      L     2;
      *D;
      T     MW 70;
      T     DB30.DBW 1;
      L     L#32768;
      <>D;
      BEC;
      L     0;
      T     MW 70;
weit: BEU;
hoch: A     M 40.3;
      L     S5T#100MS;
      SE    T 1;
      A     T 1;
      R     M 40.3;
      A     T 1;
      JC    weit;
      AN    T 1;
      S     M 40.3;
      L     MW 70;
      L     0;
      <>D;
      JC    los2;
      TAK;
      +     L#32768;
      T     MW 70;
      T     DB30.DBW 1;
      BEU;
los2: L     MW 70;
      L     2;
      /D;
      T     MW 70;
      T     DB30.DBW 1;
      L     1;
      <>D;
      BEC;
      L     0;
      T     MW 70;
      BE;
END_FUNCTION

FUNCTION FC 30 : VOID
TITLE = send
//Sends data via FDL-connection with ID=1.
//Starting at byte 1 from DB30, 4 bytes are going to send.
VERSION : 0.0
BEGIN
NETWORK
TITLE =
      O     M 50.0;
      ON    M 50.0;
      S     M 50.0;
      CALL  "AG_SEND" (
           $1                       := P#M 50.0,
           $2                       := 1,
           $3                       := 272,
           $4                       := P#DB30.DBX 1.0 BYTE 240,
           $5                       := 4,
           $6                       := M 1.2,
           $7                       := M 1.3,
           $8                       := P#M 200.0);	//AG_SEND
      BE;
END_FUNCTION

FUNCTION FC 31 : VOID
TITLE = Emfangen/Receive
//Receives data via FDL-connection with ID=1.
//Data are accepted in DB31.
VERSION : 0.0
BEGIN
NETWORK
TITLE =
      CALL  "AG_RECV" (
           $1                       := 1,
           $2                       := 272,
           $3                       := P#DB31.DBX 1.0 BYTE 240,
           $4                       := P#M 1.0,
           $5                       := M 1.1,
           $6                       := P#M 202.0,
           $7                       := P#M 10.0);	//AG_RECV
      L     DB31.DBW 1;
      T     QW 0;
      BE;
END_FUNCTION

ORGANIZATION_BLOCK OB 1
TITLE = co-ordination
//Co-ordination of the program sequence.
VERSION : 0.1
VAR_TEMP
  OB1_EV_CLASS : BYTE ;	//Bits 0-3 = 1 (Coming event), Bits 4-7 = 1 (Event class 1)
  OB1_SCAN_1 : BYTE ;	//1 (Cold restart scan 1 of OB 1), 3 (Scan 2-n of OB 1)
  OB1_PRIORITY : BYTE ;	//1 (Priority of 1 is lowest)
  OB1_OB_NUMBR : BYTE ;	//1 (Organization block 1, OB1)
  OB1_RESERVED_1 : BYTE ;	//Reserved for system
  OB1_RESERVED_2 : BYTE ;	//Reserved for system
  OB1_PREV_CYCLE : INT ;	//Cycle time of previous OB1 scan (milliseconds)
  OB1_MIN_CYCLE : INT ;	//Minimum cycle time of OB1 (milliseconds)
  OB1_MAX_CYCLE : INT ;	//Maximum cycle time of OB1 (milliseconds)
  OB1_DATE_TIME : DATE_AND_TIME ;	//Date and time OB1 started
END_VAR
BEGIN
NETWORK
TITLE =
      CALL  FC 29;
      CALL  FC 30;
      CALL  FC 31;
      BE;
END_ORGANIZATION_BLOCK

ORGANIZATION_BLOCK OB 100
TITLE = Create DB
//Creation of data blocks DB30 and DB31. The process values are saved in these 
//data blocks.
VERSION : 0.0
VAR_TEMP
  OB100_EV_CLASS : BYTE ;	//16#13, Event class 1, Entering event state, Event logged in diagnostic buffer
  OB100_STRTUP : BYTE ;	//16#81/82/83/84 Method of startup
  OB100_PRIORITY : BYTE ;	//27 (Priority of 1 is lowest)
  OB100_OB_NUMBR : BYTE ;	//100 (Organization block 100, OB100)
  OB100_RESERVED_1 : BYTE ;	//Reserved for system
  OB100_RESERVED_2 : BYTE ;	//Reserved for system
  OB100_STOP : WORD ;	//Event that caused CPU to stop (16#4xxx)
  OB100_STRT_INFO : DWORD ;	//Information on how system started
  OB100_DATE_TIME : DATE_AND_TIME ;	//Date and time OB100 started
END_VAR
BEGIN
NETWORK
TITLE =
      L     30;
      T     MW 22;
      L     31;
      T     MW 24;
      L     350;
      T     MW 26;
      CALL  SFC 22 (
           LOW_LIMIT                := MW 22,
           UP_LIMIT                 := MW 24,
           COUNT                    := MW 26,
           RET_VAL                  := MW 28,
           DB_NUMBER                := MW 30);
      CALL  SFC 22 (
           LOW_LIMIT                := MW 22,
           UP_LIMIT                 := MW 24,
           COUNT                    := MW 26,
           RET_VAL                  := MW 28,
           DB_NUMBER                := MW 30);
      BE;
END_ORGANIZATION_BLOCK

SYMBOL_TABLE
"Server variables"	DB 1	DB 1
"observe Variables"	VAT 1	
END_SYMBOL_TABLE

DATA_BLOCK "Server variables"	// DB 1
VERSION : 0.1
  STRUCT
   Index_100 : INT ;
   Index_101 : ARRAY  [1 .. 10 ] OF BYTE ;
   Index_102 : STRUCT
    Subindex_1 : BOOL ;
    Subindex_2 : STRING  [8 ] := 'Hello!!!';
    Subindex_3 : CHAR ;
    Subindex_4 : DINT ;
   END_STRUCT ;
  END_STRUCT ;	
BEGIN
   Index_102.Subindex_2 := 'Hallo!!!';
   Index_102.Subindex_3 := ' ';
END_DATA_BLOCK

ORGANIZATION_BLOCK OB 1
VERSION : 0.1
VAR_TEMP
  OB1_EV_CLASS : BYTE ;	//Bits 0-3 = 1 (Coming event), Bits 4-7 = 1 (Event class 1)
  OB1_SCAN_1 : BYTE ;	//1 (Cold restart scan 1 of OB 1), 3 (Scan 2-n of OB 1)
  OB1_PRIORITY : BYTE ;	//1 (Priority of 1 is lowest)
  OB1_OB_NUMBR : BYTE ;	//1 (Organization block 1, OB1)
  OB1_RESERVED_1 : BYTE ;	//Reserved for system
  OB1_RESERVED_2 : BYTE ;	//Reserved for system
  OB1_PREV_CYCLE : INT ;	//Cycle time of previous OB1 scan (milliseconds)
  OB1_MIN_CYCLE : INT ;	//Minimum cycle time of OB1 (milliseconds)
  OB1_MAX_CYCLE : INT ;	//Maximum cycle time of OB1 (milliseconds)
  OB1_DATE_TIME : DATE_AND_TIME ;	//Date and time OB1 started
END_VAR
BEGIN
// (block stored without names or comments; labels and parameter names are numbered)
END_ORGANIZATION_BLOCK

SYMBOL_TABLE
"DP_SEND"	FC 1	FC 1	// DP SEND
"DP_RECV"	FC 2	FC 2	// DP RECEIVE
"DP_DIAG"	FC 3	FC 3	// DP DIAGNOSE
"DP_CTRL"	FC 4	FC 4	// DP CONTROL
"WR_REC"	SFC 58	SFC 58	// Write Data Record
"RD_REC"	SFC 59	SFC 59	// Read a Data Record
END_SYMBOL_TABLE

// FC 1: know-how protected block, not included

// FC 2: know-how protected block, not included

// FC 3: know-how protected block, not included

// FC 4: know-how protected block, not included

FUNCTION FC 29 : VOID
TITLE = handle the process data
//A data word is incremented and decremented cyclically. The time intervall for 
//incrementing and decrementing is 3 seconds.
VERSION : 0.1
BEGIN
NETWORK
TITLE =
      A     T 4;	//time downwards
      JC    runt;
st_1: A     M 40.1;	//start timer 3
      L     S5T#3S;	//LED upwards 3 sec.
      SE    T 3;
      A     T 3;
      R     M 40.1;
      JC    hoch;	//jump to upwards
      AN    T 3;
      S     M 40.1;
      S     M 40.2;
runt: A     M 40.2;	//start timer 4
      L     S5T#3S;	//LED downwards 3 sec.
      SE    T 4;
      A     T 4;
      R     M 40.2;
      AN    T 4;
      S     M 40.2;
      JC    st_1;
      A     M 40.0;
      L     S5T#100MS;
      SE    T 1;
      A     T 1;
      R     M 40.0;
      A     T 1;
      JC    weit;
      AN    T 1;
      S     M 40.0;
      L     MW 70;
      L     0;
      <>D;
      JC    los1;
      TAK;
      +     1;
      T     MW 70;
      T     DB11.DBW 0;
      BEU;
los1: L     MW 70;
      L     2;
      *D;
      T     MW 70;
      T     DB11.DBW 0;
      L     L#32768;
      <>D;
      BEC;
      L     0;
      T     MW 70;
weit: BEU;
hoch: A     M 40.3;
      L     S5T#100MS;
      SE    T 1;
      A     T 1;
      R     M 40.3;
      A     T 1;
      JC    weit;
      AN    T 1;
      S     M 40.3;
      L     MW 70;
      L     0;
      <>D;
      JC    los2;
      TAK;
      +     L#32768;
      T     MW 70;
      T     DB11.DBW 0;
      BEU;
los2: L     MW 70;
      L     2;
      /D;
      T     MW 70;
      T     DB11.DBW 0;
      L     1;
      <>D;
      BEC;
      L     0;
      T     MW 70;
      BE;
END_FUNCTION

ORGANIZATION_BLOCK OB 1
TITLE = co-ordination
//Co-ordinationn of the program sequence. Calls DP_SEND and DP_RECV.
VERSION : 0.1
VAR_TEMP
  OB1_EV_CLASS : BYTE ;	//Bits 0-3 = 1 (Coming event), Bits 4-7 = 1 (Event class 1)
  OB1_SCAN_1 : BYTE ;	//1 (Cold restart scan 1 of OB 1), 3 (Scan 2-n of OB 1)
  OB1_PRIORITY : BYTE ;	//1 (Priority of 1 is lowest)
  OB1_OB_NUMBR : BYTE ;	//1 (Organization block 1, OB1)
  OB1_RESERVED_1 : BYTE ;	//Reserved for system
  OB1_RESERVED_2 : BYTE ;	//Reserved for system
  OB1_PREV_CYCLE : INT ;	//Cycle time of previous OB1 scan (milliseconds)
  OB1_MIN_CYCLE : INT ;	//Minimum cycle time of OB1 (milliseconds)
  OB1_MAX_CYCLE : INT ;	//Maximum cycle time of OB1 (milliseconds)
  OB1_DATE_TIME : DATE_AND_TIME ;	//Date and time OB1 started
END_VAR
BEGIN
NETWORK
TITLE =
      CALL  "DP_SEND" (
           $1                       := 272,
           $2                       := P#DB11.DBX 0.0 BYTE 10,
           $3                       := M 1.2,
           $4                       := M 1.3,
           $5                       := P#M 206.0);	//DP_SEND
      CALL  FC 29;
      CALL  "DP_RECV" (
           $1                       := 272,
           $2                       := P#DB10.DBX 0.0 BYTE 10,
           $3                       := P#M 1.0,
           $4                       := M 1.1,
           $5                       := P#M 200.0,
           $6                       := P#M 202.0);	//DP_RECV
      L     DB10.DBW 0;	//from DP-Slave received data
      T     QW 0;	//output to simulation module
      BE;
END_ORGANIZATION_BLOCK

ORGANIZATION_BLOCK OB 100
TITLE = create DB
//Creation of data blocks DB10 and DB11. The process values are saved in these 
//data blocks.
VERSION : 0.0
VAR_TEMP
  OB100_EV_CLASS : BYTE ;	//16#13, Event class 1, Entering event state, Event logged in diagnostic buffer
  OB100_STRTUP : BYTE ;	//16#81/82/83/84 Method of startup
  OB100_PRIORITY : BYTE ;	//27 (Priority of 1 is lowest)
  OB100_OB_NUMBR : BYTE ;	//100 (Organization block 100, OB100)
  OB100_RESERVED_1 : BYTE ;	//Reserved for system
  OB100_RESERVED_2 : BYTE ;	//Reserved for system
  OB100_STOP : WORD ;	//Event that caused CPU to stop (16#4xxx)
  OB100_STRT_INFO : DWORD ;	//Information on how system started
  OB100_DATE_TIME : DATE_AND_TIME ;	//Date and time OB100 started
END_VAR
BEGIN
NETWORK
TITLE =
      L     10;
      T     MW 20;
      L     11;
      T     MW 22;
      L     300;
      T     MW 24;
      CALL  SFC 22 (
           LOW_LIMIT                := MW 20,
           UP_LIMIT                 := MW 22,
           COUNT                    := MW 24,
           RET_VAL                  := MW 26,
           DB_NUMBER                := MW 26);
      CALL  SFC 22 (
           LOW_LIMIT                := MW 20,
           UP_LIMIT                 := MW 22,
           COUNT                    := MW 24,
           RET_VAL                  := MW 26,
           DB_NUMBER                := MW 28);
      BE;
END_ORGANIZATION_BLOCK

SYMBOL_TABLE
"AG_SEND"	FC 5	FC 5	// AG SEND
"AG_RECV"	FC 6	FC 6	// AG RECEIVE
END_SYMBOL_TABLE

// FC 5: know-how protected block, not included

// FC 6: know-how protected block, not included

FUNCTION FC 30 : VOID
TITLE = Send
//Return the data as job confirmation.
VERSION : 0.0
BEGIN
NETWORK
TITLE =
      O     M 50.0;
      ON    M 50.0;
      S     M 50.0;
      CALL  "AG_SEND" (
           $1                       := P#M 50.0,
           $2                       := 1,
           $3                       := 272,
           $4                       := P#DB31.DBX 1.0 BYTE 240,
           $5                       := 4,
           $6                       := M 1.2,
           $7                       := M 1.3,
           $8                       := P#M 200.0);	//Call AG_SEND
      BE;
END_FUNCTION

FUNCTION FC 31 : VOID
TITLE = Receive
//Save the received data in the data block and output the data to the process 
//simulation.
VERSION : 0.0
BEGIN
NETWORK
TITLE =
//Data is accepted in DB31.
      CALL  "AG_RECV" (
           $1                       := 1,
           $2                       := 272,
           $3                       := P#DB31.DBX 1.0 BYTE 240,
           $4                       := P#M 1.0,
           $5                       := M 1.1,
           $6                       := P#M 202.0,
           $7                       := P#M 10.0);	//Call AG_RECV
      L     DB31.DBW 1;
      T     QW 0;
      BE;
END_FUNCTION

ORGANIZATION_BLOCK OB 1
TITLE = co-ordination
//Co-ordination of the program sequence.
VERSION : 0.1
VAR_TEMP
  OB1_EV_CLASS : BYTE ;	//Bits 0-3 = 1 (Coming event), Bits 4-7 = 1 (Event class 1)
  OB1_SCAN_1 : BYTE ;	//1 (Cold restart scan 1 of OB 1), 3 (Scan 2-n of OB 1)
  OB1_PRIORITY : BYTE ;	//1 (Priority of 1 is lowest)
  OB1_OB_NUMBR : BYTE ;	//1 (Organization block 1, OB1)
  OB1_RESERVED_1 : BYTE ;	//Reserved for system
  OB1_RESERVED_2 : BYTE ;	//Reserved for system
  OB1_PREV_CYCLE : INT ;	//Cycle time of previous OB1 scan (milliseconds)
  OB1_MIN_CYCLE : INT ;	//Minimum cycle time of OB1 (milliseconds)
  OB1_MAX_CYCLE : INT ;	//Maximum cycle time of OB1 (milliseconds)
  OB1_DATE_TIME : DATE_AND_TIME ;	//Date and time OB1 started
END_VAR
BEGIN
NETWORK
TITLE =
      CALL  FC 30;
      CALL  FC 31;
      BE;
END_ORGANIZATION_BLOCK

ORGANIZATION_BLOCK OB 100
TITLE = Create DB
//Creation of data blocks DB30 and DB31. The process values are saved in these 
//data blocks.
VERSION : 0.0
VAR_TEMP
  OB100_EV_CLASS : BYTE ;	//16#13, Event class 1, Entering event state, Event logged in diagnostic buffer
  OB100_STRTUP : BYTE ;	//16#81/82/83/84 Method of startup
  OB100_PRIORITY : BYTE ;	//27 (Priority of 1 is lowest)
  OB100_OB_NUMBR : BYTE ;	//100 (Organization block 100, OB100)
  OB100_RESERVED_1 : BYTE ;	//Reserved for system
  OB100_RESERVED_2 : BYTE ;	//Reserved for system
  OB100_STOP : WORD ;	//Event that caused CPU to stop (16#4xxx)
  OB100_STRT_INFO : DWORD ;	//Information on how system started
  OB100_DATE_TIME : DATE_AND_TIME ;	//Date and time OB100 started
END_VAR
BEGIN
NETWORK
TITLE =
      L     30;
      T     MW 22;
      L     31;
      T     MW 24;
      L     250;
      T     MW 26;
      CALL  SFC 22 (
           LOW_LIMIT                := MW 22,
           UP_LIMIT                 := MW 24,
           COUNT                    := MW 26,
           RET_VAL                  := MW 28,
           DB_NUMBER                := MW 30);
      CALL  SFC 22 (
           LOW_LIMIT                := MW 22,
           UP_LIMIT                 := MW 24,
           COUNT                    := MW 26,
           RET_VAL                  := MW 28,
           DB_NUMBER                := MW 30);
      BE;
END_ORGANIZATION_BLOCK
